(* CODESYS project ST_wprowadzenie_szablon.project

Project tree, tasks and I/O mapping:
  Device : CODESYS Control Win V3, CODESYS, version 3.5.20.30
    application Application
      libraries: Standard, 3.5.18.0 (System)
      task VISU_TASK (cyclic, interval 100 ms, priority 31) calls VisuElems.Visu_Prg
      task MainTask (cyclic, interval t#20ms, priority 1) calls Maiin
      visualisation Visualization
      program Main [LD]
      program POU [ST]
  libraries: Standard, 3.5.18.0 (System); VisuElemBase, * (System)
  text list GlobalTextList
*)

// Device/Application/Main
PROGRAM Main
VAR
    S1_GK, S2_GK, S3_GK: BOOL;
    S1_mono_GK, S1_bi_GK, S2_mono_GK, S2_bi_GK, S3_mono_GK, S3_bi_GK: BOOL;
    H1_GK, H2_GK, H3_GK: BOOL;
    H4_GK, H5_GK, H6_GK: BOOL;
 	
END_VAR

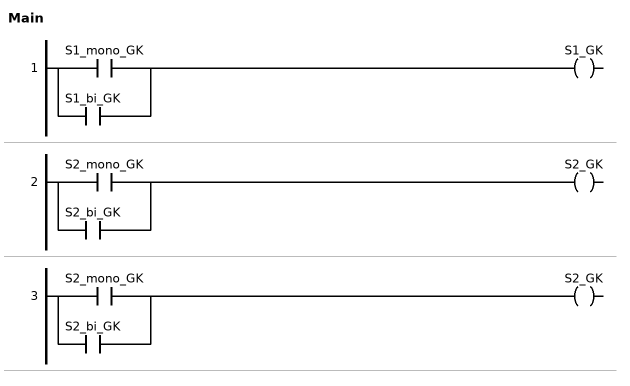
// NETWORK 1
S1_GK := S1_mono_GK OR S1_bi_GK;

// NETWORK 2
S2_GK := S2_mono_GK OR S2_bi_GK;

// NETWORK 3
S2_GK := S2_mono_GK OR S2_bi_GK;

END_PROGRAM

// Device/Application/POU
PROGRAM POU
VAR
	S1_GK, S2_GK, S3_GK: BOOL;
    S1_mono_GK, S1_bi_GK, S2_mono_GK, S2_bi_GK, S3_mono_GK, S3_bi_GK: BOOL;
    H1_GK, H2_GK, H3_GK: BOOL;
    H4_GK, H5_GK, H6_GK: BOOL;
END_VAR

END_PROGRAM

// Device/Application/Visualization
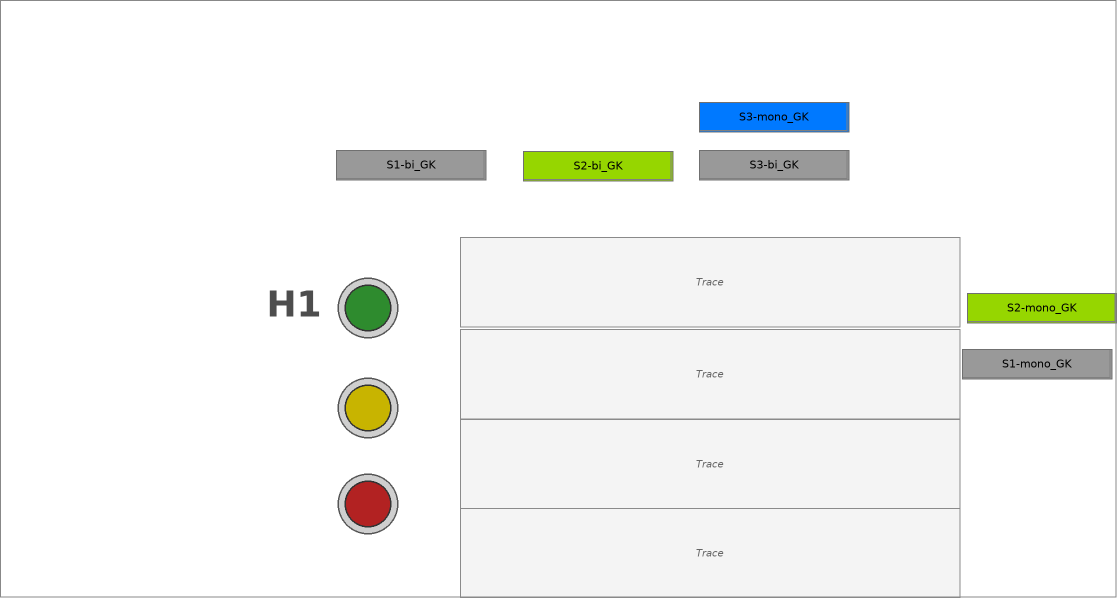
VISUALIZATION Visualization  // 1117x598
    Lamp1 (333,273 70x70), variable: Main.H1_GK, style: Lamp-Lamp1-Green
    Lamp1 (333,373 70x70), variable: Main.H2_GK, style: Lamp-Lamp1-Yellow
    Lamp1 (333,469 70x70), variable: Main.H3_GK, style: Lamp-Lamp1-Red
    Button (962,349 150x30), "S1-mono_GK"
        tap Main.S1_mono_GK
    Button (967,293 150x30), "S2-mono_GK"
        tap Main.S2_mono_GK
    Button (336,150 150x30), "S1-bi_GK"
        toggle Main.S1_bi_GK
    Button (523,151 150x30), "S2-bi_GK"
        toggle Main.S2_bi_GK
    Button (699,102 150x30), "S3-mono_GK"
        tap Main.S3_mono_GK
    Button (699,150 150x30), "S3-bi_GK"
        toggle Main.S3_bi_GK
    Trace (460,237 500x90)
    Label (219,289 150x30), "H1"
    Trace (460,329 500x90)
    Trace (460,419 500x90)
    Trace (460,508 500x90)
END_VISUALIZATION
